FUNCTION_BLOCK Signal_generator
VAR_INPUT
	T		:	TIME	:= T#2S;
END_VAR
VAR_OUTPUT
	SIGNAL	:	BOOL	:= TRUE;
END_VAR
VAR
	timer	:	TON;
END_VAR

timer(IN:= NOT timer.Q, PT:=T/2);
IF timer.Q THEN
	SIGNAL := NOT SIGNAL;
END_IF

END_FUNCTION_BLOCK

(* stored: Version 1.1.0.1, ProductVersion 3.1.4024.16
   POU Signal_generator: Id {af9d763e-313e-42be-bf5e-21670163b905}, SpecialFunc None *)
